(* IEC 61131-3 sources: sigmatek-logger-api/IXON_API/Class/IXON_LoggerAPI, 1 file *)

(* ---- IXON_LoggerAPI.st ---- *)
(*!
<Class
	Name               = "IXON_LoggerAPI"
	Revision           = "0.0"
	RealtimeTask       = "false"
	CyclicTask         = "false"
	BackgroundTask     = "false"
	Sigmatek           = "false"
	OSInterface        = "false"
	HighPriority       = "false"
	Automatic          = "false"
	UpdateMode         = "Prescan"
	SharedCommandTable = "true"
	Objectsize         = "(510,360)">
	<Channels>
		<Server Name="ClassSvr" Visualized="false" Initialize="false" WriteProtected="true" Retentive="false"/>
		<Server Name="sData" Class="IXON_LoggerAPI_Interface" Visualized="false" Initialize="false" WriteProtected="true" Retentive="false"/>
		<Server Name="sIPAddrIXON" Class="String" Visualized="true" Remotely="true" Initialize="true" WriteProtected="false" Retentive="false" Comment="use this channel to access the string functions"/>
		<Server Name="sIPAddrPLC" Class="String" Visualized="true" Remotely="true" Initialize="true" WriteProtected="false" Retentive="false" Comment="use this channel to access the string functions"/>
		<Server Name="sPasswordIXON" Class="String" Visualized="true" Remotely="true" Initialize="true" WriteProtected="false" Retentive="false" Comment="use this channel to access the string functions"/>
		<Server Name="sState" Visualized="false" Initialize="false" WriteProtected="true" Retentive="false" Comment="shows the State of the Interface Object."/>
		<Client Name="_TCPIPClient1" Required="true" Internal="true"/>
		<Client Name="MyTCPIPClient1" Required="true" Internal="true"/>
	</Channels>
	<Separators>
		<Servers>
			<SepChn Position="4"/>
			<SepChn Position="6"/>
		</Servers>
	</Separators>
	<Network Name="IXON_LoggerAPI">
		<!-- List of Components in this network -->
		<Components>
			<Object
				Name           = "_TCPIPClient1"
				Class          = "_TCPIPClient"
				Position       = "(180,150)"
				Visualized     = "true"
				Remotely       = "true"
				CyclicTime     = "10 ms"
				BackgroundTime = "always">
				<Channels>
					<Server Name="Control"/>
					<Server Name="SemaName01"/>
					<Server Name="SemaName02"/>
					<Server Name="TaskName"/>
					<Client Name="_MultiTask"/>
					<Client Name="_StdLib"/>
					<Client Name="_TaskObjectControl"/>
					<Client Name="Config"/>
					<Client Name="MaxConnections" Value="0"/>
					<Client Name="Port" Value="9230"/>
					<Client Name="SigCLib"/>
					<Client Name="SizeOfTXBuffer"/>
				</Channels>
			</Object>
			<Object
				Name       = "MyTCPIPClient1"
				Class      = "IXON_LoggerAPI_Interface"
				Position   = "(900,150)"
				Visualized = "true"
				Remotely   = "true"
				CyclicTime = "10 ms">
				<Channels>
					<Server Name="ClassSvr"/>
					<Server Name="ErrorCode"/>
					<Server Name="ErrorGroup"/>
					<Server Name="ErrorState"/>
					<Server Name="sIPAddrIXON"/>
					<Server Name="sIPAddrPLC"/>
					<Server Name="sPasswordIXON"/>
					<Server Name="sRcvCnt"/>
					<Server Name="sReconnectDelay"/>
					<Server Name="sSendDelay"/>
					<Server Name="sSndCnt"/>
					<Server Name="State"/>
					<Server Name="sTCPStep"/>
					<Client Name="_StdLib"/>
					<Client Name="_TCPIPClient"/>
				</Channels>
			</Object>
		</Components>
		<Comments>
		</Comments>
		<!-- List of Connections in this network -->
		<Connections>
			<Connection Source="this._TCPIPClient1" Destination="_TCPIPClient1.Control"/>
			<Connection Source="this.MyTCPIPClient1" Destination="MyTCPIPClient1.ClassSvr"/>
			<Connection Source="this.sIPAddrIXON" Destination="MyTCPIPClient1.sIPAddrIXON" Vertices="(1898,270),(1726,600),"/>
			<Connection Source="MyTCPIPClient1._TCPIPClient" Destination="_TCPIPClient1.Control" Vertices="(900,240),(764,240),"/>
			<Connection Source="this.sPasswordIXON" Destination="MyTCPIPClient1.sPasswordIXON" Vertices="(1898,390),(1726,720),"/>
			<Connection Source="this.sState" Destination="MyTCPIPClient1.State" Vertices="(1898,450),(1726,300),"/>
			<Connection Source="this.sIPAddrPLC" Destination="MyTCPIPClient1.sIPAddrPLC" Vertices="(1898,330),(1726,660),"/>
			<Connection Source="this.sData" Destination="MyTCPIPClient1.ClassSvr" Vertices="(1898,510),(1726,240),"/>
		</Connections>
		<!-- Headerfiles -->
		<Options>
		</Options>
	</Network>
</Class>
*)
IXON_LoggerAPI : CLASS
  //Servers:
	ClassSvr 	: SvrChCmd_DINT;
	sIPAddrIXON 	: SvrChCmd_UDINT;
	sIPAddrPLC 	: SvrChCmd_UDINT;
	sPasswordIXON 	: SvrChCmd_UDINT;
	sState 	: SvrCh__STATE_TCPIPC_INTF_PTofCls__TCPIPClientInterface;
	sData 	: SvrChCmd_DINT;
  //Clients:
	_TCPIPClient1 	: CltChCmd__TCPIPClient;
	MyTCPIPClient1 	: CltChCmd_IXON_LoggerAPI_Interface;
  //Variables:
  //Functions:

	FUNCTION VIRTUAL GLOBAL sIPAddrIXON::Read
		VAR_OUTPUT
			output (EAX) 	: UDINT;
		END_VAR;

	FUNCTION VIRTUAL GLOBAL sIPAddrIXON::Write
		VAR_INPUT
			input (EAX) 	: UDINT;
		END_VAR
		VAR_OUTPUT
			result (EAX) 	: UDINT;
		END_VAR;

	FUNCTION VIRTUAL GLOBAL sIPAddrPLC::Read
		VAR_OUTPUT
			output (EAX) 	: UDINT;
		END_VAR;

	FUNCTION VIRTUAL GLOBAL sIPAddrPLC::Write
		VAR_INPUT
			input (EAX) 	: UDINT;
		END_VAR
		VAR_OUTPUT
			result (EAX) 	: UDINT;
		END_VAR;

	FUNCTION VIRTUAL GLOBAL sPasswordIXON::Read
		VAR_OUTPUT
			output (EAX) 	: UDINT;
		END_VAR;

	FUNCTION VIRTUAL GLOBAL sPasswordIXON::Write
		VAR_INPUT
			input (EAX) 	: UDINT;
		END_VAR
		VAR_OUTPUT
			result (EAX) 	: UDINT;
		END_VAR;

	FUNCTION VIRTUAL GLOBAL sState::Read
		VAR_OUTPUT
			output (EAX) 	: _TCPIPClientInterface::_STATE_TCPIPC_INTF;
		END_VAR;

	FUNCTION VIRTUAL GLOBAL sData::Read
		VAR_OUTPUT
			output (EAX) 	: DINT;
		END_VAR;
  //Tables:
	FUNCTION @STD
		VAR_OUTPUT
			ret_code	: CONFSTATES;
		END_VAR;
	FUNCTION GLOBAL TAB @CT_;
END_CLASS;

#pragma using _TCPIPClient
#pragma using IXON_LoggerAPI_Interface

FUNCTION VIRTUAL GLOBAL IXON_LoggerAPI::sIPAddrIXON::Read
	VAR_OUTPUT
		output (EAX) 	: UDINT;
	END_VAR

	sIPAddrIXON := MyTCPIPClient1.sIPAddrIXON.Read();
	output := sIPAddrIXON;

END_FUNCTION

FUNCTION VIRTUAL GLOBAL IXON_LoggerAPI::sIPAddrIXON::Write
	VAR_INPUT
		input (EAX) 	: UDINT;
	END_VAR
	VAR_OUTPUT
		result (EAX) 	: UDINT;
	END_VAR

	sIPAddrIXON := input;
	result := (MyTCPIPClient1.sIPAddrIXON.Write(sIPAddrIXON))$UDINT;

END_FUNCTION

FUNCTION VIRTUAL GLOBAL IXON_LoggerAPI::sPasswordIXON::Read
	VAR_OUTPUT
		output (EAX) 	: UDINT;
	END_VAR

	sPasswordIXON := MyTCPIPClient1.sPasswordIXON.Read();
	output := sPasswordIXON;

END_FUNCTION

FUNCTION VIRTUAL GLOBAL IXON_LoggerAPI::sPasswordIXON::Write
	VAR_INPUT
		input (EAX) 	: UDINT;
	END_VAR
	VAR_OUTPUT
		result (EAX) 	: UDINT;
	END_VAR

	sPasswordIXON := input;
	result := (MyTCPIPClient1.sPasswordIXON.Write(sPasswordIXON))$UDINT;

END_FUNCTION

FUNCTION VIRTUAL GLOBAL IXON_LoggerAPI::sState::Read
	VAR_OUTPUT
		output (EAX) 	: _TCPIPClientInterface::_STATE_TCPIPC_INTF;
	END_VAR

	sState := MyTCPIPClient1.State.Read();
	output := sState;

END_FUNCTION

FUNCTION VIRTUAL GLOBAL IXON_LoggerAPI::sIPAddrPLC::Read
	VAR_OUTPUT
		output (EAX) 	: UDINT;
	END_VAR

	sIPAddrPLC := MyTCPIPClient1.sIPAddrPLC.Read();
	output := sIPAddrPLC;

END_FUNCTION

FUNCTION VIRTUAL GLOBAL IXON_LoggerAPI::sIPAddrPLC::Write
	VAR_INPUT
		input (EAX) 	: UDINT;
	END_VAR
	VAR_OUTPUT
		result (EAX) 	: UDINT;
	END_VAR

	sIPAddrPLC := input;
	result := (MyTCPIPClient1.sIPAddrPLC.Write(sIPAddrPLC))$UDINT;

END_FUNCTION

FUNCTION VIRTUAL GLOBAL IXON_LoggerAPI::sData::Read
	VAR_OUTPUT
		output (EAX) 	: DINT;
	END_VAR

	sData := MyTCPIPClient1.ClassSvr.Read();
	output := sData;

END_FUNCTION
